(*
Nazwa:			FB_MoveRegister
Opis:			Blok przesuniecia rejestru formatek
Wersja:			v0.3 		
Data:			2018-11-16
Autor:			DP
Urzadzenia:		 
Konfiguracja:	
Info:
- Są dwa rejestry, wejściowy i wyjsciowy (struktury)
- Jezeli rejestr ma np. 6 elementów to za kazdym razem po wykryciu trigera program będzie
	1 wejściowy przesuwał na 1 wolny (nie ma formatki) wyjściowy
	kasował 1 rejestr wejściowy
	przesuwal rejetr wejsciowy 2 na 1(przeniesiony i skasowany), 3 na 2, 4 na 3, 5 na 4, 6 na 5 i kasowal 6wejsciowy
	tym sposobem po 6 trigerach caly rejestr wejsciowy powinien być na wyjsciowym
	np po 3 trigerach na wyjsciowym powinny byc zajete 1 do 3 i na wejsciowym 1 do 3
Błędy:
1 - nie wyszło z pętli for
2 - formatka już jest w rejestrze
Uwagi:
- 
Zmiany:
2018-09-18 Dodano sprawdzanie nasadek
2018-06-14 DP Pierwsza wersja
*)

FUNCTION_BLOCK FB_MoveRegisterSortAndMoveLF
VAR_INPUT
	bFirstCycle:BOOL;					//Pierwszy cykl, zeby na początku nie wykrywało zbocza opadającego
	bTrigger :BOOL;						// Przesuniecie tablicy o jeden
	tTriggerFilterTimeOn:TIME:=T#0MS;	// Czas filtrowania wejścia Trigger na załączenie
	tTriggerFilterTimeOff:TIME:=T#0MS;	// Czas filtrowania wejścia Trigger na wyłączenie
	bTriggerBottle :BOOL;				// Zapisywanie czy jest butelka czy nie (jezeli kontrola wlączona)
	bWithBottleControl: BOOL;			// Włączona opcja kontroli butelek
	bWithCapControl:BOOL;				// Wlaczona kontrola nasadek
	bWithFormControlTrigerCounter:BOOL;	// Jezeku na trigercontrol nie ma formatki do przesunięcia to stwórz nową
	bMoveOnlyIfFormPresent:BOOL;		// Przepisuj tylko jak jest formatka
	bRotateEntranceRegisterBefore:BOOL;	// Najpierw przesuń rejestr wejściowy a następnie z niego zabierz
	bNoKeepTryingMove:BOOL;				// Dalej przepisuj jezeli nie ma miejsca
	bTriggerCap: BOOL;					// Truger wykrycia nasadki
	bReset :BOOL;						// Czyszczenie tablic
	iEntranceArrayElements :UINT; 		// Wartość koncowa tablicy
	iExitArrayElements :UINT; 			// Wartość koncowa tablicy
	bInvertWriting :BOOL;				// Wpisywanie odwrotne zamist z 1entrance na 1exit to 1entrance na 6exit	
	eClearPackageState :S_PackageState; // Czysty rejestr
END_VAR
VAR_IN_OUT
	bTriggerCounter :BOOL;		// Triger ktory jest kasowany
	eEntranceState :ARRAY [1..17] OF S_PackageState;	
	eExitState :ARRAY [1..17] OF S_PackageState;
	bKeepTryingMove :BOOL;		// Probuj dalej zapisać formatki aż się któraś zwolni
END_VAR

VAR_OUTPUT	
	bError :BOOL; 				// Błąd
	iError: UINT;				// Nr Błędu
	bTriggerDone :BOOL; 		// Wykonano przesunięcie
	bTriggerFilteredOUT:BOOL;	//Wyjscie przefiltrowanego sygnalu wejsciowego
END_VAR

VAR
	i:UINT;						// Zmienna w tablicy
	k:UINT;						// Pomocnicza zmienna do zapisywnia czy jest butelka
	rtbTrigger :R_TRIG;			// Reaguje na zbocze
	rtbTriggerBottle :R_TRIG;	// Reaguje na zbocze
	rtbReset :R_TRIG;			// Reaguje na zbocze
	TimerResetErrors :TON;		// Reset Błedu
	nFormCounter :UINT;					//Licznik formatek
	r1,r2:UINT;
	bBottlePresent: BOOL;				//Zmienna pomocnicza ze wykryto butelkę
	bCapPresent: BOOL;					//Zmienna pomocnicza ze wykryto butelkę
	j: UINT;
	tonTriggerFilterTimeOn: TON;
	bTriggerFiltered: BOOL;
	tofTriggerFilterTimeOff: TOF;
	iLFTest2: INT;
END_VAR

//Filtrowanie sygnału wejściowego
tofTriggerFilterTimeOff	(IN:=bTrigger, PT:=tTriggerFilterTimeOff);
tonTriggerFilterTimeOn	(IN:=tofTriggerFilterTimeOff.Q, PT:=tTriggerFilterTimeOn);
bTriggerFiltered 		:= tonTriggerFilterTimeOn.Q;
bTriggerFilteredOUT		:= bTriggerFiltered ;

//TRIGI I TIMERY
IF bWithBottleControl THEN
	rtbTrigger 	(CLK := NOT bTriggerFiltered, Q=>);
	rtbTriggerBottle 	(CLK := NOT bTriggerBottle, Q=>);
ELSIF bWithCapControl THEN
	rtbTrigger 	(CLK := NOT bTriggerFiltered, Q=>);
ELSE
	rtbTrigger 	(CLK := bTriggerFiltered, Q=>);
	rtbTriggerBottle 	(CLK := bTriggerBottle, Q=>);
END_IF

rtbReset 	(CLK := bReset, Q=>);
TimerResetErrors (IN:= bError, PT:=T#1000MS, Q=>);

//RESETOWANIE BLEDU
IF TimerResetErrors.Q THEN
	bError := FALSE;
END_IF

//KASOWANIE ZMIENNYCH
bTriggerDone := FALSE;

//JEZELI WLACZONO KONTROLE BUTELEK TO NADPISUJ REJESTR CZY JEST BUTELKA
IF bWithBottleControl AND bTrigger AND bTriggerBottle AND NOT bKeepTryingMove THEN //Jezeli od wykrycia formatki liczy TIMER i wykryło butelke to wpisz do rejestru że jest butelka
	eEntranceState[1].bBottlePresent := TRUE;
	eEntranceState[1].bFormPresent := TRUE;
	bBottlePresent := TRUE; // Wpisuje że jest butelka jezeli wystąpi sygnał podczas trwania czujnika formatki
ELSIF bWithBottleControl AND rtbTrigger.Q AND NOT bBottlePresent AND  NOT bKeepTryingMove AND bFirstCycle THEN
	eEntranceState[1].bBottlePresent := FALSE;
	eEntranceState[1].bFormPresent := TRUE; // jeżeli zanik czujnik formatki i nie było formatki to wpisz ze nie było butelki
END_IF
//JEZELI WLACZONO KONTROLE NASADEk TO NADPISUJ REJESTR CZY JEST BUTELKA 
(*IF bWithCapControl AND bTrigger AND bTriggerCap AND NOT bKeepTryingMove THEN //Jezeli od wykrycia formatki liczy TIMER i wykryło butelke to wpisz do rejestru że jest butelka
	eEntranceState[1].bCapPutted := TRUE;
	eEntranceState[1].bCapOK := TRUE; eEntranceState[1].bBottlePresent:= TRUE;//Zmiana nowa
	eEntranceState[1].bFormPresent := TRUE;
	bCapPresent := TRUE; // Wpisuje że jest butelka jezeli wystąpi sygnał podczas trwania czujnika formatki*)
	//ZMIANA LU 192
IF bWithCapControl AND bTriggerCap AND NOT bKeepTryingMove THEN //Jezeli od wykrycia formatki liczy TIMER i wykryło butelke to wpisz do rejestru że jest butelka
	eEntranceState[1].bCapPutted := TRUE;
	eEntranceState[1].bCapOK := TRUE; eEntranceState[1].bBottlePresent:= TRUE;//Zmiana nowa
	eEntranceState[1].bFormPresent := TRUE;
	bCapPresent := TRUE; // Wpisuje że jest butelka jezeli wystąpi sygnał podczas trwania czujnika formatki	
ELSIF bWithCapControl AND rtbTrigger.Q AND NOT bCapPresent AND  NOT bKeepTryingMove AND bFirstCycle THEN
	eEntranceState[1].bCapPutted := TRUE;
	eEntranceState[1].bCapOK:= FALSE;
	eEntranceState[1].bFormPresent := TRUE; // jeżeli zanik czujnik formatki i nie było formatki to wpisz ze nie było butelki
END_IF
//JEZELI WLACZONO SPRAWDZANIE FORMATEK Z TRIGERCOUNTER TO
IF bWithFormControlTrigerCounter  AND bTriggerCounter AND NOT bKeepTryingMove AND bFirstCycle THEN
	eEntranceState[1].bFormPresent := TRUE;
END_IF



//PRZESUNIECIE
IF (*iEntranceArrayElements <= iExitArrayElements AND*) bFirstCycle  THEN
		IF rtbTrigger.Q OR bKeepTryingMove OR bTriggerCounter THEN
		bTriggerCounter := FALSE; 
		bKeepTryingMove := FALSE;
		nFormCounter := 0;
		bBottlePresent := bCapPresent  := FALSE; 
		FOR i:= 1 TO iExitArrayElements-1 DO // SORTOWANIE
			IF NOT eExitState[i].bFormPresent THEN 
				eExitState[i] := eExitState[i+1];
				eExitState[i+1] := eClearPackageState;
			END_IF
		END_FOR

		FOR i := 1 TO iExitArrayElements DO
			IF  NOT eExitState[i].bFormPresent THEN  		// Jeżeli w rejestrze wyjściowym jest wolne miejsce to wpisz rejestr wejściowy
				
			
				eExitState[i]	:=	eEntranceState[1];			// Wpisz do rejestru dane np z [1] Buffor do [1,2,3,4,5,6] Package
				eEntranceState[1]	:=	eClearPackageState;		// Czyszczenie pierwszego rejestru wejściowego			
				k:=i;	

									// Przepisywanie zmiennej pomocniczej
				FOR i := 1 TO iEntranceArrayElements DO   				
					IF i = iEntranceArrayElements THEN
						eEntranceState[i]:=eClearPackageState;			// Zerowanie ostatniego bo zostało przesuniete wszystko o 1
					ELSE												// Przepisanie 2 do 1, 3 do 2, 4 do 3, 5 do 4, 6 do 5, zeruj 6
						eEntranceState[i] := eEntranceState[i+1]; 		// 2 do 1, 3 do 2,
						eEntranceState[i+1]:= eClearPackageState;		// zeruj 2, 
						iLFTest2:=iLFTest2;
					END_IF
				END_FOR
				
				
				
				
				bTriggerDone := TRUE;
				EXIT;
				bError := TRUE;
				iError := 5;
			ELSE
				nFormCounter := nFormCounter + 1;
				bError := TRUE;
				iError := 6;
			END_IF
		END_FOR

		IF nFormCounter = iExitArrayElements THEN
			bKeepTryingMove:=NOT bNoKeepTryingMove;
		END_IF
	END_IF
END_IF


//CZYSZCZENIE REJESTRU WEJSCIOWEGO
IF rtbReset.Q THEN
	FOR r1 := 1 TO iEntranceArrayElements DO
		eEntranceState[r1] := eClearPackageState;
	END_FOR
	FOR r2 := 1 TO iExitArrayElements DO
		eExitState[r2] := eClearPackageState;
	END_FOR
	bKeepTryingMove :=FALSE;
	bTriggerDone := FALSE;
	bTriggerCounter := FALSE; 
	nFormCounter := 0;
	bBottlePresent := bCapPresent := FALSE; 
	bError := FALSE;
	iError := 0;
END_IF

END_FUNCTION_BLOCK

(* stored: Version 1.1.0.1, ProductVersion 3.1.4026.13, FileIdentifier ada193201a185c87fa1e7e5e13ae7b625a986825, FileSignature 0bd3a4945469ecdfb20b99f5b900a15d91df146102d6fe27ef4e14d61f48a621ad7a68f9072dcb8314ffd968554310f9fdd69f2a90d4f9c98de1e3d2506d7893220702e9136749162a4c8b6adfc461bbc40082d9fd46fd7e9fedb74f78ed4f55f2f39cc9c0e7a817e370c4a7b5f06e7bb1c4fb22e242ac0d60674889b1380bf9c2207943a8a30d61853c6ccdd318f02027c59221b1d9952efe46ea560e866a2c7201dcccff3b48132fa02f6c16708eac13cfab7b9206a3325b14ba9571dd8c579b16ae77548035d03b1240ecaa8c7504317a8e97aa457308e089daa2b2a892c22b4792ab65f823ac400f4f31833cec13c0dc780d2911974031ee3a1b8fb2bc1a
   POU FB_MoveRegisterSortAndMoveLF: Id {635ae485-1441-4201-a423-ca81e330535d}, SpecialFunc None *)
